(* PLC project Unnamed, Unknown Unnamed 1 *)
(* stored: creationDateTime 2025-11-28T10:42:01, modificationDateTime 2026-02-02T15:43:14 *)

PROGRAM program0
  VAR
    Inlet : BOOL;
    WaterOutlet : BOOL;
    OilOutlet : BOOL;
    tempSensor : INT;
    levelSensor : INT := 20;
    TempReading : INT;
    LevelReading : INT;
  END_VAR

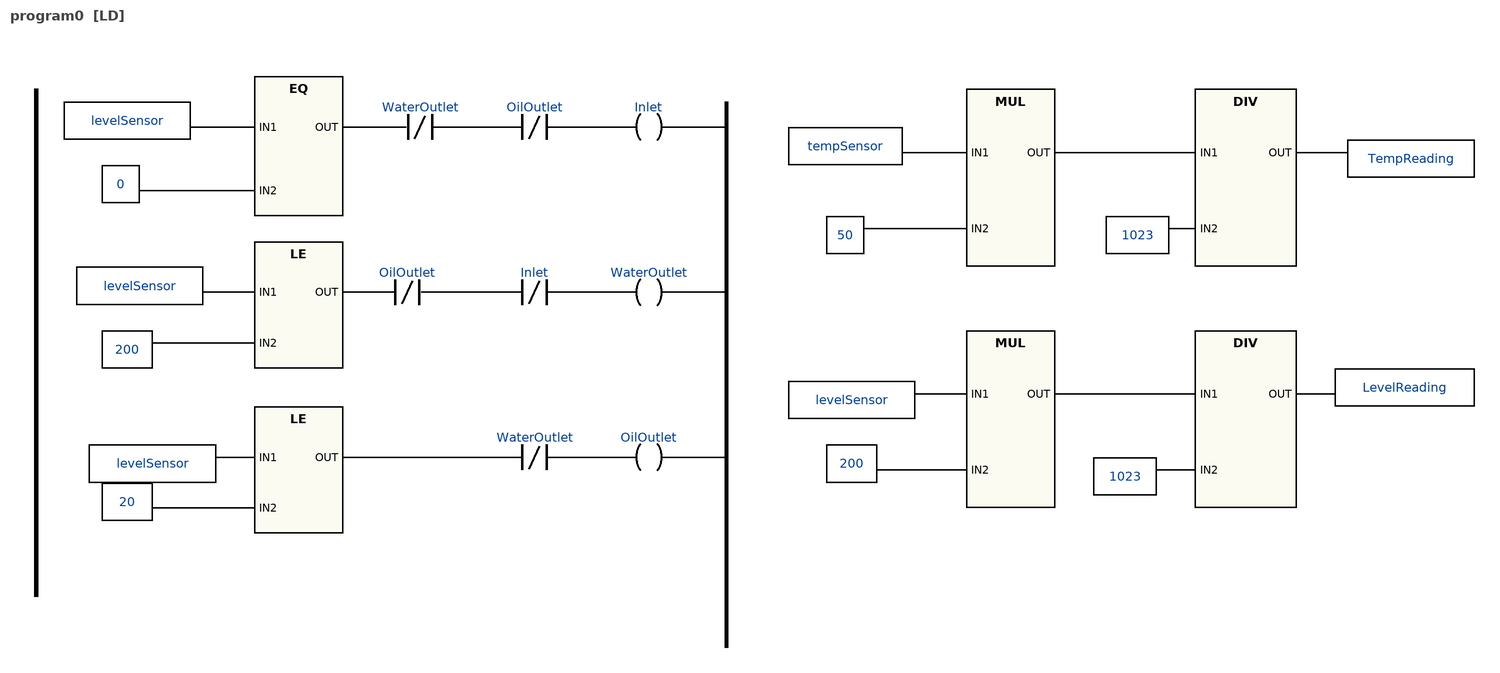
(* LD diagram, written out as Structured Text *)
TempReading := tempSensor * 50 / 1023;
LevelReading := levelSensor * 200 / 1023;
Inlet := levelSensor = 0 AND NOT WaterOutlet AND NOT OilOutlet;
OilOutlet := levelSensor <= 20 AND NOT WaterOutlet;
WaterOutlet := levelSensor <= 200 AND NOT OilOutlet AND NOT Inlet;
END_PROGRAM

CONFIGURATION Config0
  RESOURCE Res0 ON PLC
    TASK task0(INTERVAL := T#20ms, PRIORITY := 0);
    PROGRAM instance0 WITH task0 : program0;
  END_RESOURCE
END_CONFIGURATION
